INTERFACE I_Calculate

METHOD Clear : I_Calculate
END_METHOD

METHOD DecreaseBy : I_Calculate
VAR_INPUT
	lDecreaseBy : REAL;
END_VAR
END_METHOD

METHOD DivideBy : I_Calculate
VAR_INPUT
	lDivideBy : REAL;
END_VAR
END_METHOD

METHOD GetResult : LREAL
VAR_INPUT
END_VAR
END_METHOD

METHOD IncreaseBy : I_Calculate
VAR_INPUT
	lIncreaseBy : REAL;
END_VAR
END_METHOD

METHOD MultiplyBy : I_Calculate
VAR_INPUT
	lMultiplyBy : REAL;
END_VAR
END_METHOD

METHOD SetNumber : I_Calculate
VAR_INPUT
	lNumber : LREAL;
END_VAR
END_METHOD

END_INTERFACE

(* stored: Version 1.1.0.1, ProductVersion 3.1.4024.12
   Itf I_Calculate: Id {9a89b709-23b4-4f59-9523-40adfd5fa329}
   Method Clear: Id {99b54dbd-bfee-463b-ab11-2cec5955bc7d}
   Method DecreaseBy: Id {8b94408c-fd63-4aa5-b636-baf239f7028e}
   Method DivideBy: Id {71bcaa5c-b3bf-4673-8566-ac685c13bfac}
   Method GetResult: Id {3bcc4857-e052-457f-a9c1-aff1a05e935f}
   Method IncreaseBy: Id {e8644b0e-0c6d-4710-be1b-4f6c4a23f7af}
   Method MultiplyBy: Id {0b9d9e96-f758-4358-b75b-72e2c3603b98}
   Method SetNumber: Id {a2d82639-f74a-4fe7-8d71-7f8b1d0bf467} *)
